FUNCTION_BLOCK AxisControl_Encoder
VAR_INPUT
	MethodCall: BOOL;
	EmergencyStopSignal : BOOL;
	Direction : BOOL;
	EncoderStartPosition_01 : UDINT;
	EncoderStartPosition_02 : UDINT;
	EncoderTargetPosition_01 : UDINT;
	EncoderTargetPosition_02 : UDINT;	
	TouchSensor: BOOL;
	TouchSensorRelief : BOOL;
	TOF_Time_MotorControl: TIME;
	TOF_Time_TouchSensorRelief: TIME;
	AutomaticMode: BOOL;
END_VAR

VAR_OUTPUT
	MotorControl_01: BOOL;
	MotorControl_02: BOOL;
	ResetCall: BOOL;
END_VAR

VAR
//FlipFlop
	RS_AxisControl: RS;
	RS_Endschalter_Entlasten: RS;
//Zeitverzögerung
	TOF_Endschalter_Entlasten: TOF;
	TOF_MotorControl: TOF;	
//Flanke	
	R_TRIG_MethodCall: R_TRIG;
	R_TRIG_EncoderPos_01 : R_TRIG;
	R_TRIG_EncoderPos_02 : R_TRIG;

END_VAR
VAR // added by the converter: edge detectors and wires of the graphical bodies
    _w1, _w2 : BOOL;
END_VAR

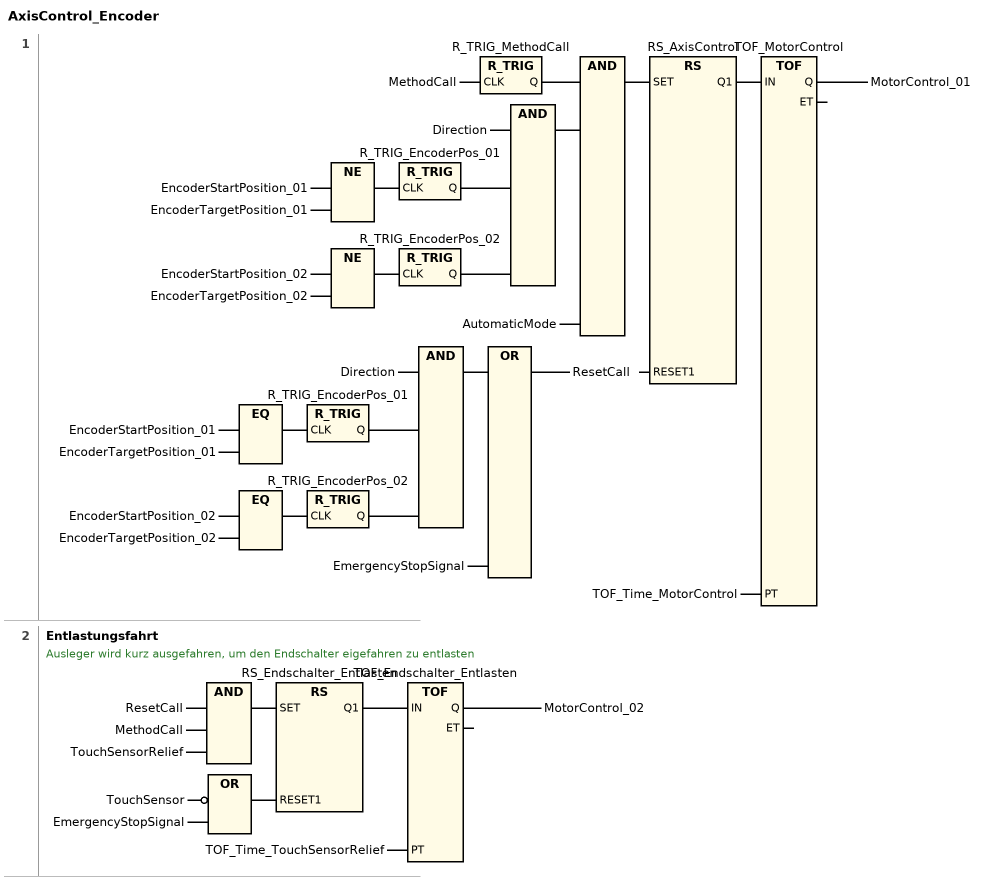
// NETWORK 1
R_TRIG_MethodCall(CLK := MethodCall); // R_TRIG
R_TRIG_EncoderPos_01(CLK := EncoderStartPosition_01 <> EncoderTargetPosition_01); // R_TRIG
R_TRIG_EncoderPos_02(CLK := EncoderStartPosition_02 <> EncoderTargetPosition_02); // R_TRIG
_w2 := R_TRIG_MethodCall.Q AND (Direction AND R_TRIG_EncoderPos_01.Q AND R_TRIG_EncoderPos_02.Q) AND AutomaticMode;
R_TRIG_EncoderPos_01(CLK := EncoderStartPosition_01 = EncoderTargetPosition_01); // R_TRIG
R_TRIG_EncoderPos_02(CLK := EncoderStartPosition_02 = EncoderTargetPosition_02); // R_TRIG
_w1 := Direction AND R_TRIG_EncoderPos_01.Q AND R_TRIG_EncoderPos_02.Q OR EmergencyStopSignal;
ResetCall := _w1;
RS_AxisControl(SET := _w2, RESET1 := _w1); // RS
TOF_MotorControl(IN := RS_AxisControl.Q1, PT := TOF_Time_MotorControl); // TOF
MotorControl_01 := TOF_MotorControl.Q;

// NETWORK 2: Entlastungsfahrt
// Ausleger wird kurz ausgefahren, um den Endschalter eigefahren zu entlasten
RS_Endschalter_Entlasten(SET := ResetCall AND MethodCall AND TouchSensorRelief, RESET1 := NOT TouchSensor OR EmergencyStopSignal); // RS
TOF_Endschalter_Entlasten(IN := RS_Endschalter_Entlasten.Q1, PT := TOF_Time_TouchSensorRelief); // TOF
MotorControl_02 := TOF_Endschalter_Entlasten.Q;

END_FUNCTION_BLOCK

(* stored: Version 1.1.0.1, ProductVersion 3.1.4024.15
   POU AxisControl_Encoder: Id {04a405fa-b8a6-44be-9c08-47c6a80a871d}, SpecialFunc None *)
